(* IEC 61131-3 sources: repolevel_ST_code_completion/real_groud_truth最新/repoeval_Builder_Application_RPI/full_result, 3 files *)

(* ---- ConcreteBuilder.st ---- *)
//This is the concrete builder class, reponsible for building the final product object
FUNCTION_BLOCK ConcreteBuilder IMPLEMENTS ITF_Builder
VAR_INPUT
END_VAR
VAR_OUTPUT
END_VAR

//Holds an internal reference to how the final product should be so the builder class can build it on the fly
//without any help from other classes excepting the Director class that is going to be passing the special specifications.
localProduct : Product;

//Stores the specifications, sent by the client, of the final product to be built.
specifications : ARRAY [1..4] OF STRING;

//Method to set the main part of the product
METHOD Set_Main_Part : VOID
VAR_INPUT
    mainPartSpec : STRING; // Specification for the main part
END_VAR
VAR_OUTPUT
END_VAR
VAR
END_VAR
THIS^.localProduct.mainPart := mainPartSpec;

//Method to set Part 1 of the product
METHOD Set_Part1 : VOID
VAR_INPUT
    part1Spec : STRING; // Specification for Part 1
END_VAR
VAR_OUTPUT
END_VAR
VAR
END_VAR
THIS^.localProduct.part1 := part1Spec;

//Method to set Part 2 of the product
METHOD Set_Part2 : VOID
VAR_INPUT
    part2Spec : STRING; // Specification for Part 2
END_VAR
VAR_OUTPUT
END_VAR
VAR
END_VAR
THIS^.localProduct.part2 := part2Spec;

//Method to set Part 3 of the product
METHOD Set_Part3 : VOID
VAR_INPUT
    part3Spec : STRING; // Specification for Part 3
END_VAR
VAR_OUTPUT
END_VAR
VAR
END_VAR
THIS^.localProduct.part3 := part3Spec;

//Method to get the final product
METHOD Get_Result : Product
VAR_INPUT
END_VAR
VAR_OUTPUT
END_VAR
VAR
END_VAR
Get_Result := THIS^.localProduct;
END_FUNCTION_BLOCK

(* ---- Director.st ---- *)
{attribute 'enable_dynamic_creation'}
//The director class is responsible to delegate the construction of the final product object
// to a concrete builder object.
FUNCTION_BLOCK Director
VAR_INPUT
	//Reference to the builder that is going to be building the final product object.
	inputConcreteBuilder : ConcreteBuilder(specs := inputConcreteBuilder.specifications);
END_VAR
VAR_OUTPUT
END_VAR

VAR
	// Holds a reference to the concrete builder object to send the specifications of the final product to it.
	concreteBuilder : ConcreteBuilder(specs := THIS^.concreteBuilder.specifications);
	// Variable to instantiate the concreteBuilder instance on the input section. It does not affect the Director's instantiation.
	defaultArray : ARRAY [1..4] OF STRING := ['Default', 'Default', 'Default', 'Default'];
END_VAR

// The Director class is responsible for delegating the construction of the final product object
// to a concrete builder object. The following methods define the behavior of the Director.

METHOD fb_init
VAR_INPUT
	// Reference to the builder that is going to be building the final product object.
	inputConcreteBuilder : ConcreteBuilder(specs := inputConcreteBuilder.specifications);
	// Necessary fields for the constructor
	bInitRetains : BOOL; // TRUE: the Retain-variables are initialized (reset warm / reset cold)
	bInCopyCode : BOOL;  // TRUE: the instance will be copied to the copy-code afterward (online change)
END_VAR
VAR_OUTPUT
END_VAR
VAR
	// Holds a reference to the concrete builder object to send the specifications of the final product to it.
	concreteBuilder : ConcreteBuilder(specs := THIS^.concreteBuilder.specifications);
END_VAR

// Initialize the Director instance by assigning the input concrete builder.
IF inputConcreteBuilder <> 0 THEN
	THIS^.concreteBuilder := inputConcreteBuilder;
ELSE
	// Assign default specifications if no input builder is provided.
	THIS^.concreteBuilder := ConcreteBuilder(specs := defaultArray);
END_IF;

// Ensure the Director is properly initialized.
fb_init := TRUE;

// Method to construct the product using the concrete builder.
METHOD Construct : Product
VAR_INPUT
	// Reference to the builder that is going to be building the final product object.
	inputConcreteBuilder : ConcreteBuilder(specs := inputConcreteBuilder.specifications);
END_VAR
VAR_OUTPUT
END_VAR
VAR
	// Holds a reference to the concrete builder object to send the specifications of the final product to it.
	concreteBuilder : ConcreteBuilder(specs := THIS^.concreteBuilder.specifications);
END_VAR

// Step-by-step construction process
// Step 1: Set the main part of the product.
THIS^.concreteBuilder.Set_Main_Part(THIS^.concreteBuilder.specifications[1]);

// Step 2: Set Part 1 of the product.
THIS^.concreteBuilder.Set_Part1(THIS^.concreteBuilder.specifications[2]);

// Step 3: Set Part 2 of the product.
THIS^.concreteBuilder.Set_Part2(THIS^.concreteBuilder.specifications[3]);

// Step 4: Set Part 3 of the product.
THIS^.concreteBuilder.Set_Part3(THIS^.concreteBuilder.specifications[4]);

// Deliver the final product.
Construct := THIS^.concreteBuilder.Get_Result();
END_FUNCTION_BLOCK

(* ---- Product.st ---- *)
{attribute 'enable_dynamic_creation'}
//The class Product is just a plain bluprint of the components of the object to be built.
//The final Product may ot may not contain the all the Parts listed on the Product declaration
// rather only the parts in the specifications sent by the client.
FUNCTION_BLOCK Product
VAR_INPUT
	//List of possible parts to be build in a final Product object
	mainPart 	: STRING;
	part1 		: STRING;
	part2 		: STRING;
	part3 		: STRING;
END_VAR
VAR_OUTPUT
END_VAR

# --------------------------------------------------
# the below code fragment can be found in:
# Builder_Application_RPI-FUN\ConcreteBuilder_Set_Part1.st (continued)
# --------------------------------------------------
# //Illustrative method of the pattern to set the part1 (continued)
# VAR
# 	//Holds an internal reference to how the final product should be so the builder class can build it on the fly
# 	// without any help from other classes excepting the Director class that is going to be passing the special
# 	// specifications to the builder.
# 	localProduct : Product;
#
# 	//Stores the specifications, sent by the client, of the final product to be built.
# 	specifications : ARRAY [1..4] OF STRING;
# END_VAR
#
# //Sets the passed value to its corresponding field.
# //We can say that the final product is in process of being built.
# //So this is a step into building the final product done by the builder.
# THIS^.localProduct.part1 := part1;

# --------------------------------------------------
# the below code fragment can be found in:
# Builder_Application_RPI-FUN\ConcreteBuilder_Build_Product.st
# --------------------------------------------------
# //Illustrative method of the pattern to build the final product
METHOD Build_Product
VAR_INPUT
END_VAR
VAR_OUTPUT
	//Returns the final product object built by the builder
	finalProduct : Product;
END_VAR
VAR
	//Holds an internal reference to how the final product should be so the builder class can build it on the fly
	// without any help from other classes excepting the Director class that is going to be passing the special
	// specifications to the builder.
	localProduct : Product;
END_VAR

//Builds the final product based on the specifications provided by the client
IF THIS^.specifications[1] <> '' THEN
	THIS^.localProduct.mainPart := THIS^.specifications[1];
END_IF

IF THIS^.specifications[2] <> '' THEN
	THIS^.localProduct.part1 := THIS^.specifications[2];
END_IF

IF THIS^.specifications[3] <> '' THEN
	THIS^.localProduct.part2 := THIS^.specifications[3];
END_IF

IF THIS^.specifications[4] <> '' THEN
	THIS^.localProduct.part3 := THIS^.specifications[4];
END_IF

//Returns the fully built product
finalProduct := THIS^.localProduct;
END_FUNCTION_BLOCK
